FUNCTION TryConvert_USINT_TO_WORD : BOOL
VAR_INPUT
	in : USINT;
	out : REFERENCE TO WORD;
END_VAR

out := USINT_TO_WORD(in);
TryConvert_USINT_TO_WORD := TRUE;

END_FUNCTION

(* stored: Version 1.1.0.1, ProductVersion 3.1.4024.12
   POU TryConvert_USINT_TO_WORD: Id {59b0e420-14b1-4233-beb0-02d1f8dcf40a}, SpecialFunc None *)
